{attribute 'no_check'}
FUNCTION_BLOCK IOMotorStarDelta
VAR_INPUT
	InAck													:	BOOL := TRUE;
	StartRight												:	BOOL := FALSE;
	FeedRight												:	BOOL := TRUE;
	PT_RestartDel											:	TIME := T#0S;
	PT_Delta												: 	TIME := T#5S;
	ProtSwitchOK											: 	FUSE;
	ProtSwitchOK2											: 	FUSE;
END_VAR                 						
VAR_OUTPUT              						
	Busy													:	BOOL;
	Error													:	BOOL;
	Status													:	BYTE;
	RestartDelActive										:	BOOL;
	ET_RestartDel											: 	TIME;	(* waiting-time of start interlock *)
END_VAR                 						
VAR                     						
	TON_StarDelta											:	TON;
	TP_RestartDel											:	TP;
	_StarContactor									AT %Q* 	: 	BOOL;
	_DeltaContactor									AT %Q* 	: 	BOOL;
	_MainContactor									AT %Q* 	: 	BOOL;
END_VAR

(* Start Delta Motor IO	 				 	V1.1	*)
(****************************************************)

(* Protection Switch *****************************************)
	IF InAck 
	THEN 
		Ack(); 
	END_IF

	ProtSwitchOK(
		Force	:= ,
		Invert	:= ,
		InAck 	:= FALSE,
		Q		=> ,
		Event	=> ,
		INPUT 	=> );

	ProtSwitchOK2(InAck 	:= FALSE);
	
(* Start ****************************************************)
	IF StartRight THEN
		_MainContactor 										:= 	NOT TP_RestartDel.Q
																AND ProtSwitchOK.Q 
																AND ProtSwitchOK2.Q	
																AND FeedRight;
                       										
		_StarContactor 										:= 	_MainContactor
																AND NOT TON_StarDelta.Q
																AND NOT _DeltaContactor;

		_DeltaContactor 									:= 	_MainContactor
																AND TON_StarDelta.Q;

		TP_RestartDel();
	ELSE
		TP_RestartDel(IN := _MainContactor , PT := PT_RestartDel);
		_MainContactor 										:= FALSE;
		_DeltaContactor 									:= FALSE;
		_StarContactor 										:= FALSE;
	END_IF

(* Timer *****************************************************)
	TON_StarDelta( IN := _MainContactor, PT := PT_Delta);

(* Status ***********************************************************)
	Busy	 												:= _MainContactor;
	Error													:= NOT ProtSwitchOK.Q OR NOT ProtSwitchOK2.Q; 
	RestartDelActive										:= TP_RestartDel.Q;
	
	IF TP_RestartDel.ET > T#0MS 
	THEN
		ET_RestartDel		:= TP_RestartDel.PT - TP_RestartDel.ET;
	ELSE
		ET_RestartDel		:= t#0ms;
	END_IF
	
(* HmiStatus **************************************************)
	Status.0												 := NOT _MainContactor;
	Status.1												 := _MainContactor;
	Status.2												 := _DeltaContactor;
	Status.3												 := RestartDelActive;
	Status.4												 := FALSE;
	Status.5												 := FeedRight;
	Status.6												 := NOT Error AND NOT RestartDelActive;
	Status.7												 := Error;

(*********************************************************************)

METHOD PUBLIC Ack
VAR_INPUT
END_VAR
ProtSwitchOK(InAck := TRUE);
ProtSwitchOK2(InAck := TRUE);
END_METHOD

METHOD PUBLIC Reset
VAR_INPUT
END_VAR
Ack();
SetStop();
END_METHOD

METHOD PUBLIC ResetRestartTmr
VAR_INPUT
END_VAR
MEMSET(ADR(TP_RestartDel),0,SIZEOF(TP_RestartDel));
END_METHOD

METHOD PUBLIC SetStartRight
VAR_INPUT
END_VAR
StartRight 													:= TRUE;
END_METHOD

METHOD PUBLIC SetStop
VAR_INPUT
END_VAR
StartRight 													:= FALSE;
_MainContactor 												:= FALSE;
_DeltaContactor 											:= FALSE;
_StarContactor 												:= FALSE;
END_METHOD

END_FUNCTION_BLOCK

(* stored: Version 1.1.0.1, ProductVersion 3.1.4024.12
   POU IOMotorStarDelta: Id {5594a7dd-ad46-4be3-a1e3-b417ee472759}, SpecialFunc None
   Method Ack: Id {5caacf8f-eac6-4896-8ee5-6c07cd6f77d1}
   Method Reset: Id {76803435-65ad-48dc-91c1-f4f2ff360476}
   Method ResetRestartTmr: Id {75d4b8cc-d3b2-45a2-8101-3838b9dde8c9}
   Method SetStartRight: Id {ee358356-0117-4719-be9d-cfeeaf9c337b}
   Method SetStop: Id {58ac8580-5271-4843-bf3b-95c144bab2be} *)
